ABB RobotStudio station: Lab1Part3.rspag

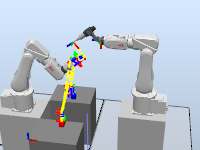
--- station ---
Station Lab1Part3_4 (saved by RobotStudio 7.0.8732.594)
Controller Controller1, task T_ROB2: task frame (RAPID world) sits at (-600, 0, 500) mm in the station
Controller Controller1, task T_ROB1: task frame (RAPID world) sits at (-600, 0, 500) mm in the station
Controller Controller1
  mechanical unit ROB_1: obj_robot, 6 joints, base frame (0, 0, 0) mm
  mechanical unit ROB_2: tool_robot, 6 joints, base frame (1100, 0, 100) mm, rotated rx 0 ry 0 rz 180 deg
Layout (positions relative to the parent item):
  - ObjTable [part] at (-100, 0, 0) mm
  - ToolRobot [part] at (200, 0, 0) mm
  - Table2 [part]
  - Table1 [part]
  - tool_robot [mechanism, from Robots\IRB120_3_58_G_01.rslib] at (500, 0, 600) mm, rotated rx 0 ry 0 rz 180 deg; joint values [0, 0, 0, 0, 0, 0] (rad or m)
  - obj_robot [mechanism, from Robots\IRB120_3_58_G_01.rslib] at (-600, 0, 500) mm; joint values [0.1601, 0.3735, 0.4749, -0.012, -1.5485, 0.0047] (rad or m)
  - Smart_Gripper_Servo_Fingers [mechanism, from Libraries\Smart_Gripper_Servo_Fingers.rslib] at (-199.55, 65.56, 907.5) mm, rotated rx -0.39 ry 49.89 rz 9.57 deg; joint values [0.025] (rad or m)
  - BlueCube [part]
  - MyTool_4 [mechanism, from Training Objects\myTool.rslib] at (126, 0, 1230) mm, rotated rx 0 ry 90 rz -180 deg
  - GreenCube [part]
  - RedCube [part]
Attachment: Smart_Gripper_Servo_Fingers is attached to obj_robot / Link6
Attachment: MyTool_4 is attached to tool_robot / Link6
EventTableEntry 2775: Group=, Trigger=Gripper 2776, Actions=[EventTableActionMechanicalPose 2777, EventTableActionAttach 2778], Comment=, ActivationMode=2, Cyclic=false
EventTableTriggerIO 2776: IOValue=[1], IRC5Controller=? -1, Operator=0, SignalSource=Controller1 1565
EventTableActionMechanicalPose 2777: VirtualSignal=, Mechanism=Smart_Gripper_Servo_Fingers 1548, ToPoseName=SyncPosition, VirtualSignalValue=[1]
EventTableActionAttach 2778: AttachmentParent=Smart_Gripper_Servo_Fingers 1548, AttachmentChild=? -1, MountObject=false, Offset=[X=1, Y=0, Z=0, W=0, X=0, Y=1, Z=0, W=0, X=0, Y=0, Z=1, W=0, X=0, Y=0, Z=0, W=1], FlangeIndext=0, FindNearest=true
EventTableEntry 2779: Group=, Trigger=Gripper 2780, Actions=[EventTableActionMechanicalPose 2781, EventTableActionDetach 2782], Comment=, ActivationMode=2, Cyclic=false
EventTableTriggerIO 2780: IOValue=[0], IRC5Controller=? -1, Operator=0, SignalSource=Controller1 1565
EventTableActionMechanicalPose 2781: VirtualSignal=, Mechanism=Smart_Gripper_Servo_Fingers 1548, ToPoseName=HomePosition, VirtualSignalValue=[1]
EventTableActionDetach 2782: AttachmentParent=Smart_Gripper_Servo_Fingers 1548, AttachmentChild=? -1
Targets, tools, work objects and paths stored in the station and not in the controller backup, written as RAPID:
! task T_ROB1
MODULE Module1
  VAR SyncIdent Ident_1;
  VAR SyncIdent Ident_2;
  VAR SyncIdent Ident_3;
  VAR SyncIdent Ident_4;
  VAR SyncIdent Ident_5;
  VAR SyncIdent Ident_6;
  VAR SyncIdent Ident_7;
  VAR SyncIdent Ident_8;
  VAR SyncIdent Ident_9;
  VAR SyncIdent Ident_10;
ENDMODULE

! task T_ROB2
MODULE Module1
  VAR SyncIdent Ident_1;
  VAR SyncIdent Ident_2;
  VAR SyncIdent Ident_3;
  VAR SyncIdent Ident_4;
  VAR SyncIdent Ident_5;
  VAR SyncIdent Ident_6;
  VAR SyncIdent Ident_7;
  VAR SyncIdent Ident_8;
  VAR SyncIdent Ident_9;
  VAR SyncIdent Ident_10;
ENDMODULE


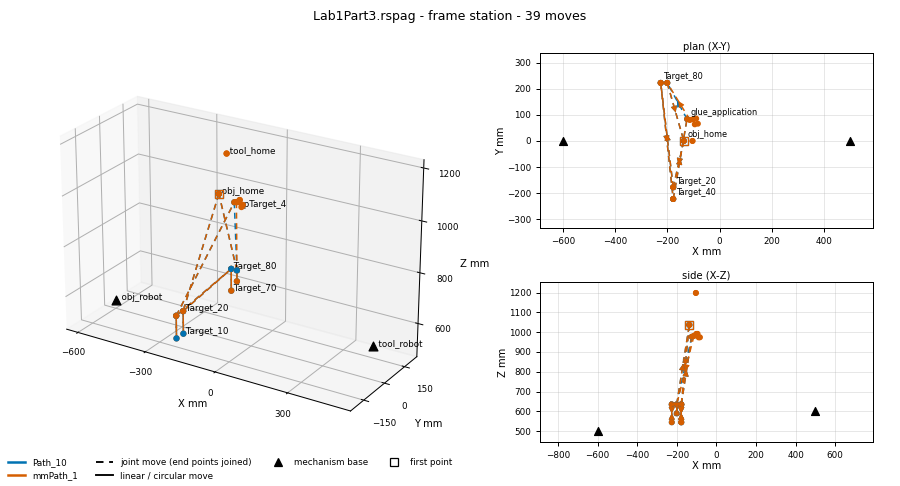
[picture p0: tool path of Lab1Part3.rspag in frame station, 39 of 60 moves have a stored position in this frame; points joined in program order, loops and branches not executed]
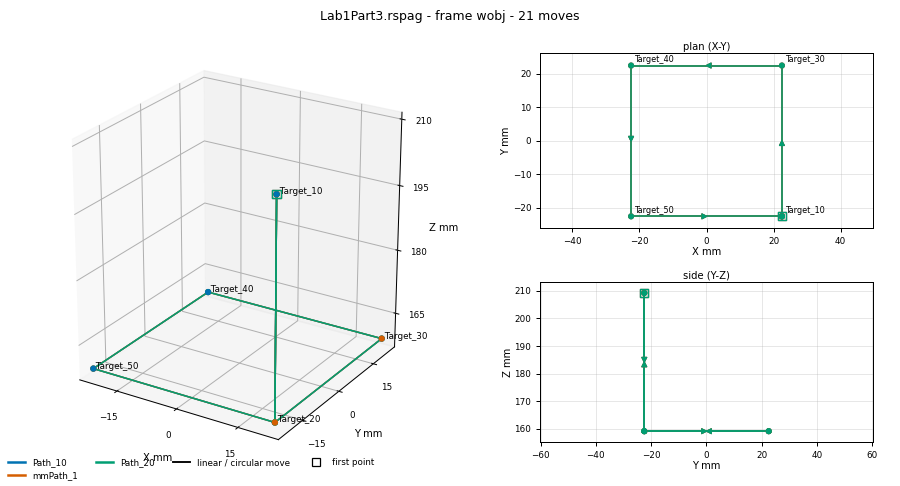
[picture p1: tool path of Lab1Part3.rspag in frame wobj, 21 of 60 moves have a stored position in this frame; points joined in program order, loops and branches not executed]
--- Backups/Controller1/RAPID/TASK1/PROGMOD/CalibData.mod ---
MODULE CalibData
	PERS tooldata Servo:=[TRUE,[[0,0,114.2],[1,0,0,0]],[0.215,[8.7,12.3,49.2],[1,0,0,0],0.00021,0.00024,0.00009]];
	TASK PERS wobjdata wobj:=[FALSE,TRUE,"",[[200,-450,0],[1,0,0,0]],[[0,0,0],[1,0,0,0]]];
ENDMODULE

--- Backups/Controller1/RAPID/TASK1/PROGMOD/Module1.mod ---
MODULE Module1
	CONST robtarget obj_home:=[[463.253930185,0,536.9],[0.5,0,0.866025404,0],[0,0,0,0],[9E+09,9E+09,9E+09,9E+09,9E+09,9E+09]];
	CONST robtarget Target_20:=[[222.5,272.5,135],[0,0,1,0],[-1,0,-1,0],[9E+09,9E+09,9E+09,9E+09,9E+09,9E+09]];
	CONST robtarget Target_10:=[[222.5,272.5,45],[0,0,1,0],[-1,0,-1,0],[9E+09,9E+09,9E+09,9E+09,9E+09,9E+09]];
	CONST robtarget Target_80:=[[174.5,672.5,135],[0,0,1,0],[0,0,0,0],[9E+09,9E+09,9E+09,9E+09,9E+09,9E+09]];
	CONST robtarget Target_70:=[[174.5,672.5,45],[0,0,1,0],[0,0,0,0],[9E+09,9E+09,9E+09,9E+09,9E+09,9E+09]];
	CONST robtarget Target_40:=[[222.5,227.5,135],[0,0,1,0],[-1,0,-1,0],[9E+09,9E+09,9E+09,9E+09,9E+09,9E+09]];
	CONST robtarget Target_30:=[[222.5,227.5,45],[0,0,1,0],[-1,0,-1,0],[9E+09,9E+09,9E+09,9E+09,9E+09,9E+09]];
	CONST robtarget glue_application:=[[475.394161922,83.824817218,477.053771392],[0.902859012,-0.036833609,0.421010072,0.078989928],[0,-1,0,1],[9E+09,9E+09,9E+09,9E+09,9E+09,9E+09]];
	VAR syncident Ident_1;
	PERS tasks Task_1{2}:=[["T_ROB1"],["T_ROB2"]];
	CONST robtarget pTarget_1:=[[486.140132177,80.74651396,481.57609232],[0.903372542,-0.037303746,0.419791766,0.079381068],[0,-1,0,1],[9E+09,9E+09,9E+09,9E+09,9E+09,9E+09]];
	CONST robtarget pTarget_2:=[[498.795178743,83.036821461,491.441203872],[0.905529452,-0.042240307,0.413294177,0.086139953],[0,-1,0,1],[9E+09,9E+09,9E+09,9E+09,9E+09,9E+09]];
	CONST robtarget pTarget_3:=[[505.053878761,63.607308475,491.778526777],[0.906832849,-0.029989912,0.414732667,0.068931877],[0,-1,0,1],[9E+09,9E+09,9E+09,9E+09,9E+09,9E+09]];
	CONST robtarget pTarget_4:=[[516.951065525,66.013890202,474.138314916],[0.896165035,-0.034082598,0.436465715,0.072279223],[0,-1,0,1],[9E+09,9E+09,9E+09,9E+09,9E+09,9E+09]];
	CONST robtarget pTarget_5:=[[510.575607298,85.72642658,473.668582687],[0.894895314,-0.046932896,0.434896823,0.08845583],[0,-1,0,1],[9E+09,9E+09,9E+09,9E+09,9E+09,9E+09]];
	CONST robtarget pTarget_6:=[[499.084273507,83.119879708,490.97407041],[0.905565927,-0.043157613,0.413613075,0.083737664],[0,-1,0,1],[9E+09,9E+09,9E+09,9E+09,9E+09,9E+09]];
	CONST robtarget pTarget_7:=[[486.441923635,80.838638203,481.068225135],[0.903428469,-0.038235803,0.420020381,0.077057805],[0,-1,0,1],[9E+09,9E+09,9E+09,9E+09,9E+09,9E+09]];
	VAR syncident Ident_2;
	CONST robtarget Target_100:=[[199.5,672.5,135],[0,0,1,0],[0,0,0,0],[9E+09,9E+09,9E+09,9E+09,9E+09,9E+09]];
	CONST robtarget Target_90:=[[199.5,672.5,90],[0,0,1,0],[0,0,0,0],[9E+09,9E+09,9E+09,9E+09,9E+09,9E+09]];
	VAR syncident Ident_6;
	VAR syncident Ident_5;
	VAR syncident Ident_7;
	VAR syncident Ident_8;
	VAR syncident Ident_9;
	VAR syncident Ident_10;
    !***********************************************************
    !
    ! Module:  Module1
    !
    ! Description:
    !   <Insert description here>
    !
    ! Author: bruno
    !
    ! Version: 1.0
    !
    !***********************************************************


    !***********************************************************
    !
    ! Procedure main
    !
    !   This is the entry point of your program
    !
    !***********************************************************
    PROC main()
        !Add your code here
    ENDPROC
	PROC Path_10()
	    Reset Gripper;
	    MoveJ obj_home,v60,z5,Servo\WObj:=wobj0;
	    MoveJ Target_20,v60,z5,Servo\WObj:=wobj;
	    MoveJ Target_10,v60,z5,Servo\WObj:=wobj;
	    WaitTime\InPos,1;
	    Set Gripper;
	    MoveJ Target_20,v60,z5,Servo\WObj:=wobj;
	    MoveJ Target_80,v60,z5,Servo\WObj:=wobj;
	    MoveJ Target_70,v60,z5,Servo\WObj:=wobj;
	    WaitTime\InPos,1;
	    Reset Gripper;
		MoveJ Target_80,v60,z5,Servo\WObj:=wobj;
		MoveJ Target_40,v60,z5,Servo\WObj:=wobj;
		MoveJ Target_30,v60,z5,Servo\WObj:=wobj;
		WaitTime\InPos,1;
		Set Gripper;
		MoveJ Target_40,v60,z5,Servo\WObj:=wobj;
		MoveJ glue_application,v60,z5,Servo\WObj:=wobj0;
		WaitTime\InPos,1;
		Reset Gripper;
		MoveJ Target_100,v60,z5,Servo\WObj:=wobj;
		MoveJ Target_90,v60,z5,Servo\WObj:=wobj;
		WaitTime\InPos,1;
		Reset Gripper;
		MoveJ Target_100,v60,z5,Servo\WObj:=wobj;
		MoveJ obj_home,v60,z5,Servo\WObj:=wobj0;
	ENDPROC
	PROC mmPath_1()
	    Reset Gripper;
	    MoveJ obj_home,v60,fine,Servo\WObj:=wobj0;
	    MoveJ Target_20,v60,fine,Servo\WObj:=wobj;
	    MoveJ Target_10,v60,fine,Servo\WObj:=wobj;
	    WaitTime\InPos,1;
	    Set Gripper;
	    MoveJ Target_20,v60,fine,Servo\WObj:=wobj;
	    MoveJ Target_80,v60,fine,Servo\WObj:=wobj;
	    MoveJ Target_70,v60,fine,Servo\WObj:=wobj;
	    WaitTime\InPos,1;
	    Reset Gripper;
	    MoveJ Target_80,v60,fine,Servo\WObj:=wobj;
	    MoveJ Target_40,v60,fine,Servo\WObj:=wobj;
	    MoveJ Target_30,v60,fine,Servo\WObj:=wobj;
	    WaitTime\InPos,1;
	    Set Gripper;
	    MoveJ Target_40,v60,fine,Servo\WObj:=wobj;
	    MoveJ glue_application,v60,fine,Servo\WObj:=wobj0;
	    WaitTime\InPos,1;
	    SyncMoveOn Ident_9,Task_1;
	    MoveL pTarget_1\ID:=10,v60,fine,Servo\WObj:=wobj0;
	    MoveL pTarget_2\ID:=20,v60,fine,Servo\WObj:=wobj0;
	    MoveL pTarget_3\ID:=30,v60,fine,Servo\WObj:=wobj0;
	    MoveL pTarget_4\ID:=40,v60,fine,Servo\WObj:=wobj0;
	    MoveL pTarget_5\ID:=50,v60,fine,Servo\WObj:=wobj0;
	    MoveL pTarget_6\ID:=60,v60,fine,Servo\WObj:=wobj0;
	    MoveL pTarget_7\ID:=70,v60,fine,Servo\WObj:=wobj0;
	    SyncMoveOff Ident_10;
		MoveJ Target_100,v60,fine,Servo\WObj:=wobj;
		MoveJ Target_90,v60,fine,Servo\WObj:=wobj;
		WaitTime\InPos,1;
		Reset Gripper;
		MoveJ Target_100,v60,fine,Servo\WObj:=wobj;
		MoveJ obj_home,v60,fine,Servo\WObj:=wobj0;
	ENDPROC
	PROC Path_20()

	ENDPROC
ENDMODULE

--- Backups/Controller1/RAPID/TASK2/PROGMOD/CalibData.mod ---
MODULE CalibData
	PERS tooldata MyTool:=[TRUE,[[31.792631019,0,229.638935148],[0.945518576,0,0.325568154,0]],[1,[0,0,1],[1,0,0,0],0,0,0]];
	TASK PERS wobjdata wobj:=[FALSE,FALSE,"ROB_1",[[527.492191753,70.163879046,488.743],[0.262004394,-0.719842834,0.604024939,-0.21984964]],[[0,0,0],[1,0,0,0]]];
ENDMODULE

--- Backups/Controller1/RAPID/TASK2/PROGMOD/Module1.mod ---
MODULE Module1
	CONST robtarget Target_10:=[[22.499988517,-22.499993257,209.200000349],[0.00000006,-0.707106774,0.707106788,0.000000057],[0,0,0,0],[9E+09,9E+09,9E+09,9E+09,9E+09,9E+09]];
	CONST robtarget Target_20:=[[22.499996754,-22.499993078,159.200000348],[0.00000006,-0.707106774,0.707106788,0.000000057],[0,0,0,0],[9E+09,9E+09,9E+09,9E+09,9E+09,9E+09]];
	CONST robtarget Target_30:=[[22.499997703,22.500006921,159.200000509],[0.00000006,-0.707106774,0.707106788,0.000000057],[0,0,0,0],[9E+09,9E+09,9E+09,9E+09,9E+09,9E+09]];
	CONST robtarget Target_40:=[[-22.500002297,22.500007871,159.199993095],[0.000000059,-0.707106774,0.707106788,-0.000000057],[0,0,0,0],[9E+09,9E+09,9E+09,9E+09,9E+09,9E+09]];
	CONST robtarget Target_50:=[[-22.500003246,-22.49999213,159.199992935],[0.00000006,-0.707106774,0.707106788,-0.000000057],[0,0,0,0],[9E+09,9E+09,9E+09,9E+09,9E+09,9E+09]];
	CONST robtarget Target_60:=[[22.499996754,-22.499993078,159.200000348],[0.000000057,-0.707106774,0.707106788,-0.000000059],[0,0,0,0],[9E+09,9E+09,9E+09,9E+09,9E+09,9E+09]];
	CONST robtarget Target_70:=[[22.499988517,-22.499993257,209.200000349],[0.000000057,-0.707106774,0.707106788,-0.000000059],[0,0,0,0],[9E+09,9E+09,9E+09,9E+09,9E+09,9E+09]];
	VAR syncident Ident_1;
	PERS tasks Task_1{2}:=[["T_ROB1"],["T_ROB2"]];
	CONST robtarget pTarget_1:=[[22.499988517,-22.499993257,209.200000349],[0.00000006,-0.707106774,0.707106788,0.000000057],[0,-1,1,0],[9E+09,9E+09,9E+09,9E+09,9E+09,9E+09]];
	CONST robtarget pTarget_2:=[[22.499996754,-22.499993078,159.200000348],[0.00000006,-0.707106774,0.707106788,0.000000057],[0,-1,1,0],[9E+09,9E+09,9E+09,9E+09,9E+09,9E+09]];
	CONST robtarget pTarget_3:=[[22.499997703,22.500006921,159.200000509],[0.00000006,-0.707106774,0.707106788,0.000000057],[0,-1,1,0],[9E+09,9E+09,9E+09,9E+09,9E+09,9E+09]];
	CONST robtarget pTarget_4:=[[-22.500002297,22.500007871,159.199993095],[0.000000059,-0.707106774,0.707106788,-0.000000057],[0,-1,1,0],[9E+09,9E+09,9E+09,9E+09,9E+09,9E+09]];
	CONST robtarget pTarget_5:=[[-22.500003246,-22.49999213,159.199992935],[0.00000006,-0.707106774,0.707106788,-0.000000057],[0,-1,1,0],[9E+09,9E+09,9E+09,9E+09,9E+09,9E+09]];
	CONST robtarget pTarget_6:=[[22.499996754,-22.499993078,159.200000348],[0.000000057,-0.707106774,0.707106788,-0.000000059],[0,-1,1,0],[9E+09,9E+09,9E+09,9E+09,9E+09,9E+09]];
	CONST robtarget pTarget_7:=[[22.499988517,-22.499993257,209.200000349],[0.000000057,-0.707106774,0.707106788,-0.000000059],[0,-1,1,0],[9E+09,9E+09,9E+09,9E+09,9E+09,9E+09]];
	VAR syncident Ident_2;
	VAR syncident Ident_6;
	VAR syncident Ident_5;
	VAR syncident Ident_8;
	VAR syncident Ident_7;
	VAR syncident Ident_10;
	VAR syncident Ident_9;
	CONST robtarget tool_home:=[[496.361064852,0,698.207368981],[0,0.898794046,0,-0.438371147],[0,0,0,0],[9E+09,9E+09,9E+09,9E+09,9E+09,9E+09]];
    !***********************************************************
    !
    ! Module:  Module1
    !
    ! Description:
    !   <Insert description here>
    !
    ! Author: bruno
    !
    ! Version: 1.0
    !
    !***********************************************************


    !***********************************************************
    !
    ! Procedure main
    !
    !   This is the entry point of your program
    !
    !***********************************************************
    PROC main()
        !Add your code here
    ENDPROC
	PROC Path_10()
	    MoveL Target_10,v60,fine,MyTool\WObj:=wobj;
	    MoveL Target_20,v60,fine,MyTool\WObj:=wobj;
	    MoveL Target_30,v60,fine,MyTool\WObj:=wobj;
	    MoveL Target_40,v60,fine,MyTool\WObj:=wobj;
	    MoveL Target_50,v60,fine,MyTool\WObj:=wobj;
	    MoveL Target_60,v60,fine,MyTool\WObj:=wobj;
	    MoveL Target_70,v60,fine,MyTool\WObj:=wobj;
	ENDPROC
	PROC mmPath_1()
	    MoveJ tool_home,v60,fine,MyTool\WObj:=wobj0;
	    SyncMoveOn Ident_9,Task_1;
	    MoveJ pTarget_1\ID:=10,v60,fine,MyTool\WObj:=wobj;
	    MoveL pTarget_2\ID:=20,v60,fine,MyTool\WObj:=wobj;
	    MoveL pTarget_3\ID:=30,v60,fine,MyTool\WObj:=wobj;
	    MoveL pTarget_4\ID:=40,v60,fine,MyTool\WObj:=wobj;
	    MoveL pTarget_5\ID:=50,v60,fine,MyTool\WObj:=wobj;
	    MoveL pTarget_6\ID:=60,v60,fine,MyTool\WObj:=wobj;
	    MoveL pTarget_7\ID:=70,v60,fine,MyTool\WObj:=wobj;
	    SyncMoveOff Ident_10;
		MoveJ tool_home,v60,fine,MyTool\WObj:=wobj0;
	ENDPROC
	PROC Path_20()
	    MoveL Target_10,v60,fine,MyTool\WObj:=wobj;
	    MoveL Target_20,v60,fine,MyTool\WObj:=wobj;
	    MoveL Target_30,v60,fine,MyTool\WObj:=wobj;
	    MoveL Target_40,v60,fine,MyTool\WObj:=wobj;
	    MoveL Target_50,v60,fine,MyTool\WObj:=wobj;
	    MoveL Target_60,v60,fine,MyTool\WObj:=wobj;
	    MoveL Target_70,v60,fine,MyTool\WObj:=wobj;
	ENDPROC
ENDMODULE

--- Backups/Controller1/SYSPAR/EIO.cfg ---
EIO:CFG_1.0:6:1::
#
EIO_SIGNAL:

      -Name "Gripper" -SignalType "DO" -Access "All"
